{attribute 'qualified_only'}
{attribute 'strict'}
{attribute 'to_string'}
TYPE enum_FB_ESTOP :
(
	undefine := 0,
	run := 1,
	stop := 2,
	safe := 3,
	error := 4,
	reset :=  5,
	start := 6,
	delayout := 8
);
END_TYPE

(* stored: Version 1.1.0.1
   DUT enum_FB_ESTOP: Id {e765f3c7-07f7-4e7f-8c81-3d5fab92f5c5} *)
